TYPE aS_AnalogAlarm :
STRUCT
	HIHI: REAL;
	HI: REAL;
	LO: REAL;
	LOLO: REAL;
	Deadband: REAL;
END_STRUCT
END_TYPE

(* stored: Version 1.1.0.1, ProductVersion 3.1.4024.4
   DUT aS_AnalogAlarm: Id {17efecf2-f00c-4de0-ad2f-f9fb71c1ebb7} *)
